// TIA Portal project "TankFillingSystem" (V15)

(* hardware
DEVICE "S7-1200 station_1"  S7-1200 Station
   slot 0: "Rack_0"  S7-1200 Rack  Rack  V1.0
   slot 1: "Filling System Controller"  CPU 1214C DC/DC/DC  6ES7 214-1AG40-0XB0  V4.2
      slot 3: "AQ 1x12BIT_1"  AQ1 signal board  6ES7 232-4HA30-0XB0  V1.0
   slot 101: "CM 1243-5"  CM 1243-5  6GK7 243-5DX30-0XE0  V1.3
   slot 102: "CM 1241 (RS485)_1"  CM 1241 (RS485)  6ES7 241-1CH30-0XB0  V1.0
*)

// ===== PLC "Filling System Controller"  CPU 1214C DC/DC/DC =====

VAR_GLOBAL   // PLC tag table "Default tag table"
   "START" AT %I0.0 : Bool;
   "WORK" AT %M0.0 : Bool;
   "Bottom_Sensor1" AT %I0.1 : Bool;
   "Top_Sensor1" AT %I0.2 : Bool;
   "Tank1_Low_Level" AT %Q0.0 : Bool;
   "Tank1_Medium_Level" AT %Q0.1 : Bool;
   "Tank1_High_Level" AT %Q0.2 : Bool;
   "Tank1_Malfunction" AT %Q0.3 : Bool;
   "malfunction_Tank1_Edge" AT %M100.0 : Bool;
   "Tank1_Malfunction_Memory" AT %M200.0 : Bool;
   "MemoryClock1Hz" AT %M50.5 : Bool;
   "Confirm" AT %I0.6 : Bool;
   "Emergency_Channel_Generator_Edge" AT %M101.0 : Bool;
   "Emergency_Channel_Malfuncion_Memory" AT %M101.1 : Bool;
   "Emergency_Channel_Malfunction_Edge" AT %M101.2 : Bool;
   "Valve_Control" AT %I0.3 : Bool;
   "Valve_Status" AT %Q0.4 : Bool;
   "Pump_Status" AT %Q0.5 : Bool;
   "STOP" AT %I0.7 : Bool;
   "Liquid_Motion_Generator" AT %M20.0 : Bool;
END_VAR

DATA_BLOCK "Tank1_DB"   // DB1
{ S7_Optimized_Access := 'TRUE' }
VERSION : 0.1
// stored: InstanceOfName Tank
"Tank"
BEGIN
   Capacity := 1000.0;
   Fill_Level := 1000.0;
   Growth := ;
END_DATA_BLOCK

DATA_BLOCK "Pump_DB"   // DB2
{ S7_Optimized_Access := 'TRUE' }
VERSION : 0.1
// stored: InstanceOfName Pump
"Pump"
BEGIN
   Growth := 2.5;
END_DATA_BLOCK

FUNCTION_BLOCK "Tank"   // FB1, LAD
TITLE = Tank
{ S7_Optimized_Access := 'TRUE' }
VERSION : 0.1
// The logic for signalization of liquid level in the tank
   VAR_INPUT
      Botom_Level_Sensor : Bool;   // Bottom level sensor reading
      Top_Level_Sensor : Bool;   // Top level sensor reading
      Valve_Control : Bool;   // Valve control - open / close
   END_VAR
   VAR_OUTPUT
      Low_Level : Bool;   // The liquid is at the low level in tank
      Medium_Level : Bool;   // The liquid is at the medium level in tank
      High_Level : Bool;   // The liquid is at the high level in tank
      Malfunction : Bool;   // Malfunction: tank is leaning
      Valve_Status : Bool;   // Output infromation about valve status is open or closed
   END_VAR
   VAR
      Capacity : Real;   // Tank capacity
      Fill_Level : Real;   // Current fill level of liquid
      Valve_Remote : Bool;   // Valve remote controlling
      Generator_Edge : Bool;
      Growth : Real;   // how fill level decrease
   END_VAR
   VAR_TEMP   // added for the SCL form of the ladder/FBD networks
      _w1 : Bool;
   END_VAR
BEGIN

REGION Network 1: the liquid is at the low level in tank
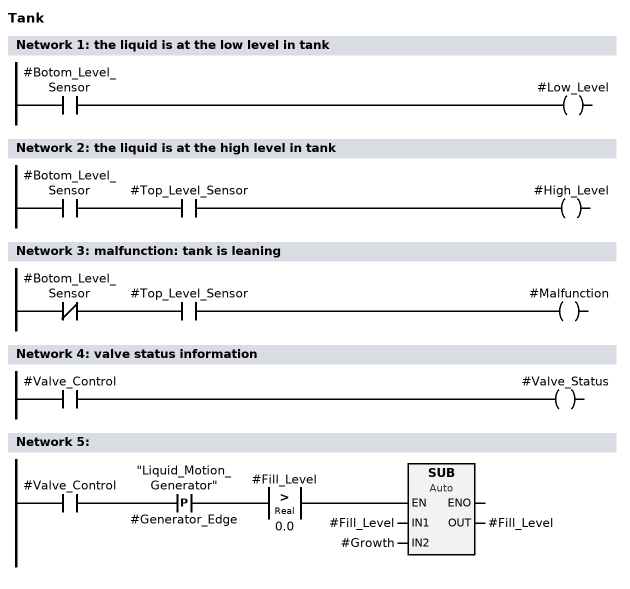
   RUNG wire#powerrail
      Contact( #Botom_Level_Sensor )
      Coil( #Low_Level )
   END_RUNG
   // the same network as SCL:
   #Low_Level := #Botom_Level_Sensor;
END_REGION

REGION Network 2: the liquid is at the high level in tank
   RUNG wire#powerrail
      Contact( #Botom_Level_Sensor )
      Contact( #Top_Level_Sensor )
      Coil( #High_Level )
   END_RUNG
   // the same network as SCL:
   #High_Level := #Botom_Level_Sensor AND #Top_Level_Sensor;
END_REGION

REGION Network 3: malfunction: tank is leaning
   RUNG wire#powerrail
      I_Contact( #Botom_Level_Sensor )
      Contact( #Top_Level_Sensor )
      Coil( #Malfunction )
   END_RUNG
   // the same network as SCL:
   #Malfunction := NOT #Botom_Level_Sensor AND #Top_Level_Sensor;
END_REGION

REGION Network 4: valve status information
   RUNG wire#powerrail
      Contact( #Valve_Control )
      Coil( #Valve_Status )
   END_RUNG
   // the same network as SCL:
   #Valve_Status := #Valve_Control;
END_REGION

REGION Network 5
   RUNG wire#powerrail
      Contact( #Valve_Control )
      P_Contact(operand := "Liquid_Motion_Generator", bit := #Generator_Edge)
      { S7_Templates := "SrcType := Real" } GT_Contact(in1 := #Fill_Level, in2 := 0.0)
      Sub(in1 := #Fill_Level, in2 := #Growth, out => #Fill_Level)
   END_RUNG
   // the same network as SCL:
   #_w1 := #Valve_Control AND "Liquid_Motion_Generator" AND NOT #Generator_Edge;   // rising edge of "Liquid_Motion_Generator"
   #Generator_Edge := "Liquid_Motion_Generator";
   IF #_w1 AND (#Fill_Level > 0.0) THEN #Fill_Level := #Fill_Level - #Growth; END_IF;
END_REGION
END_FUNCTION_BLOCK

FUNCTION_BLOCK "Pump"   // FB2, LAD
TITLE = Pump
{ S7_Optimized_Access := 'TRUE' }
VERSION : 0.1
// Logic of pump controlling
   VAR_INPUT
      Low_Level : Bool;   // Liquid level is at low
      Top_Level : Bool;   // Liquid level is at top
      Malfunction : Bool;   // Tank malfunction input information
      Capacity : Real;   // Tank capacity
   END_VAR
   VAR_OUTPUT
      Work_Status : Bool;   // pump is working
   END_VAR
   VAR_IN_OUT
      FillLevel : Real;
   END_VAR
   VAR
      Growth : Real;   // value of fill level increase
      Work : Bool;
      Generator_Edge : Bool;
   END_VAR
   VAR_TEMP   // added for the SCL form of the ladder/FBD networks
      _w1 : Bool;
   END_VAR
BEGIN

REGION Network 1: pump is working
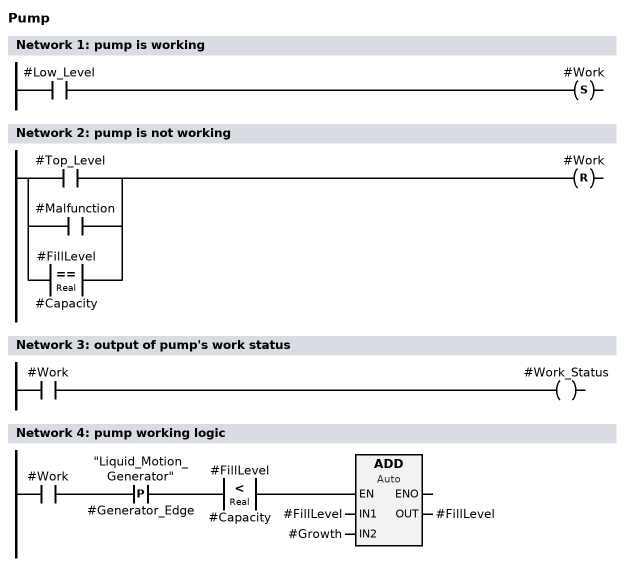
   RUNG wire#powerrail
      Contact( #Low_Level )
      S_Coil( #Work )
   END_RUNG
   // the same network as SCL:
   IF #Low_Level THEN #Work := TRUE; END_IF;
END_REGION

REGION Network 2: pump is not working
   RUNG wire#powerrail
      Contact( #Top_Level )
      wire#w1
      R_Coil( #Work )
   END_RUNG
   RUNG wire#powerrail
      Contact( #Malfunction )
   END_RUNG wire#w1
   RUNG wire#powerrail
      { S7_Templates := "SrcType := Real" } EQ_Contact(in1 := #FillLevel, in2 := #Capacity)
   END_RUNG wire#w1
   // the same network as SCL:
   IF #Top_Level OR #Malfunction OR (#FillLevel = #Capacity) THEN #Work := FALSE; END_IF;
END_REGION

REGION Network 3: output of pump's work status
   RUNG wire#powerrail
      Contact( #Work )
      Coil( #Work_Status )
   END_RUNG
   // the same network as SCL:
   #Work_Status := #Work;
END_REGION

REGION Network 4: pump working logic
   RUNG wire#powerrail
      Contact( #Work )
      P_Contact(operand := "Liquid_Motion_Generator", bit := #Generator_Edge)
      { S7_Templates := "SrcType := Real" } LT_Contact(in1 := #FillLevel, in2 := #Capacity)
      Add(in1 := #FillLevel, in2 := #Growth, out => #FillLevel)
   END_RUNG
   // the same network as SCL:
   #_w1 := #Work AND "Liquid_Motion_Generator" AND NOT #Generator_Edge;   // rising edge of "Liquid_Motion_Generator"
   #Generator_Edge := "Liquid_Motion_Generator";
   IF #_w1 AND (#FillLevel < #Capacity) THEN #FillLevel := #FillLevel + #Growth; END_IF;
END_REGION
END_FUNCTION_BLOCK

FUNCTION "EmergencyChannel" : Void   // FC1, LAD
{ S7_Optimized_Access := 'TRUE' }
VERSION : 0.1
   VAR_INPUT
      Hardware_Generator : Bool;   // Hardware Generator for flashing sygnalization
      Confirm : Bool;   // Malfunction confirming
      Malfunction : Bool;   // information about occured malfunction
   END_VAR
   VAR_OUTPUT
      Malfunction_Signal : Bool;   // the signalization of occured malfunction: flashing, continous
   END_VAR
   VAR_IN_OUT
      Generator_Edge : Bool;   // Hardware Generator edge memory
      Malfunction_Memory : Bool;   // memory that store information about malfunction in the previous circle
      Malfunction_Edge : Bool;   // The Rising edge for malfunction input signal
   END_VAR
   VAR_TEMP   // added for the SCL form of the ladder/FBD networks
      _w1 : Bool;
   END_VAR
BEGIN

REGION Network 1: memory that store information about malfunction in the previous circle
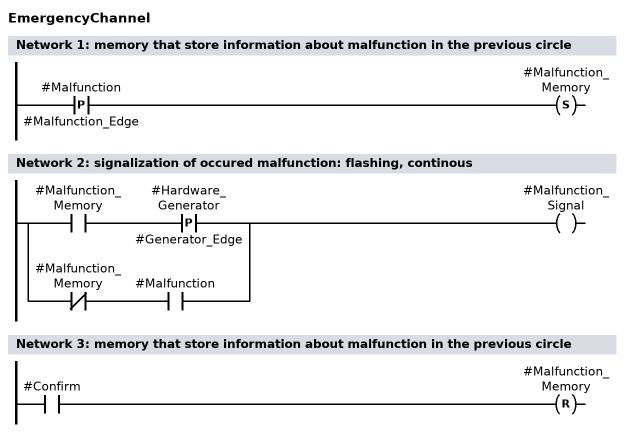
   RUNG wire#powerrail
      P_Contact(operand := #Malfunction, bit := #Malfunction_Edge)
      S_Coil( #Malfunction_Memory )
   END_RUNG
   // the same network as SCL:
   #_w1 := #Malfunction AND NOT #Malfunction_Edge;   // rising edge of #Malfunction
   #Malfunction_Edge := #Malfunction;
   IF #_w1 THEN #Malfunction_Memory := TRUE; END_IF;
END_REGION

REGION Network 2: signalization of occured malfunction: flashing, continous
   RUNG wire#powerrail
      Contact( #Malfunction_Memory )
      P_Contact(operand := #Hardware_Generator, bit := #Generator_Edge)
      wire#w1
      Coil( #Malfunction_Signal )
   END_RUNG
   RUNG wire#powerrail
      I_Contact( #Malfunction_Memory )
      Contact( #Malfunction )
   END_RUNG wire#w1
   // the same network as SCL:
   #_w1 := #Malfunction_Memory AND #Hardware_Generator AND NOT #Generator_Edge;   // rising edge of #Hardware_Generator
   #Generator_Edge := #Hardware_Generator;
   #Malfunction_Signal := #_w1 OR (NOT #Malfunction_Memory AND #Malfunction);
END_REGION

REGION Network 3: memory that store information about malfunction in the previous circle
   RUNG wire#powerrail
      Contact( #Confirm )
      R_Coil( #Malfunction_Memory )
   END_RUNG
   // the same network as SCL:
   IF #Confirm THEN #Malfunction_Memory := FALSE; END_IF;
END_REGION
END_FUNCTION

ORGANIZATION_BLOCK "Main"   // OB1, LAD, ProgramCycle
TITLE = "Main Program Sweep (Cycle)"
{ S7_Optimized_Access := 'TRUE' }
VERSION : 0.1
   VAR_INPUT
      Initial_Call : Bool;   // Initial call of this OB
      Remanence : Bool;   // =True, if remanent data are available
   END_VAR
BEGIN

REGION Network 1
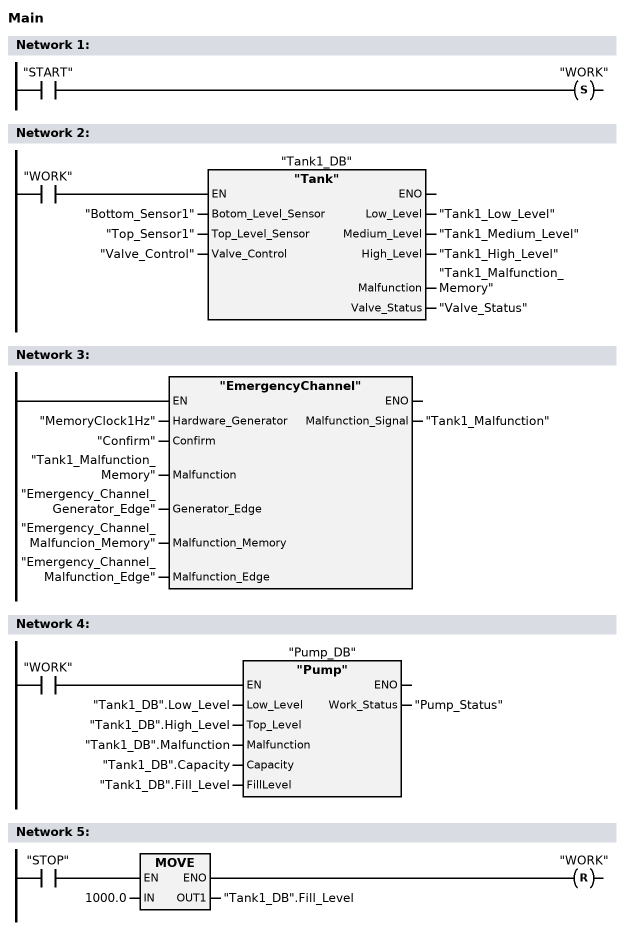
   RUNG wire#powerrail
      Contact( "START" )
      S_Coil( "WORK" )
   END_RUNG
   // the same network as SCL:
   IF "START" THEN "WORK" := TRUE; END_IF;
END_REGION

REGION Network 2
   RUNG wire#powerrail
      Contact( "WORK" )
      "Tank1_DB"(Botom_Level_Sensor := "Bottom_Sensor1", Top_Level_Sensor := "Top_Sensor1", Valve_Control := "Valve_Control", Low_Level => "Tank1_Low_Level", Medium_Level => "Tank1_Medium_Level", High_Level => "Tank1_High_Level", Malfunction => "Tank1_Malfunction_Memory", Valve_Status => "Valve_Status")
   END_RUNG
   // the same network as SCL:
   IF "WORK" THEN
       "Tank1_DB"(Botom_Level_Sensor := "Bottom_Sensor1",   // "Tank"
                  Top_Level_Sensor := "Top_Sensor1",
                  Valve_Control := "Valve_Control",
                  Low_Level => "Tank1_Low_Level",
                  Medium_Level => "Tank1_Medium_Level",
                  High_Level => "Tank1_High_Level",
                  Malfunction => "Tank1_Malfunction_Memory",
                  Valve_Status => "Valve_Status");
   END_IF;
END_REGION

REGION Network 3
   RUNG wire#powerrail
      "EmergencyChannel"(Hardware_Generator := "MemoryClock1Hz", Confirm := "Confirm", Malfunction := "Tank1_Malfunction_Memory", Generator_Edge := "Emergency_Channel_Generator_Edge", Malfunction_Memory := "Emergency_Channel_Malfuncion_Memory", Malfunction_Edge := "Emergency_Channel_Malfunction_Edge", Malfunction_Signal => "Tank1_Malfunction")
   END_RUNG
   // the same network as SCL:
   "EmergencyChannel"(Hardware_Generator := "MemoryClock1Hz",
                      Confirm := "Confirm",
                      Malfunction := "Tank1_Malfunction_Memory",
                      Generator_Edge := "Emergency_Channel_Generator_Edge",
                      Malfunction_Memory := "Emergency_Channel_Malfuncion_Memory",
                      Malfunction_Edge := "Emergency_Channel_Malfunction_Edge",
                      Malfunction_Signal => "Tank1_Malfunction");
END_REGION

REGION Network 4
   RUNG wire#powerrail
      Contact( "WORK" )
      "Pump_DB"(Low_Level := "Tank1_DB".Low_Level, Top_Level := "Tank1_DB".High_Level, Malfunction := "Tank1_DB".Malfunction, Capacity := "Tank1_DB".Capacity, FillLevel := "Tank1_DB".Fill_Level, Work_Status => "Pump_Status")
   END_RUNG
   // the same network as SCL:
   IF "WORK" THEN
       "Pump_DB"(Low_Level := "Tank1_DB".Low_Level,   // "Pump"
                 Top_Level := "Tank1_DB".High_Level,
                 Malfunction := "Tank1_DB".Malfunction,
                 Capacity := "Tank1_DB".Capacity,
                 FillLevel := "Tank1_DB".Fill_Level,
                 Work_Status => "Pump_Status");
   END_IF;
END_REGION

REGION Network 5
   RUNG wire#powerrail
      Contact( "STOP" )
      Move(in := 1000.0, out1 => "Tank1_DB".Fill_Level)
      R_Coil( "WORK" )
   END_RUNG
   // the same network as SCL:
   IF "STOP" THEN
       "Tank1_DB".Fill_Level := 1000.0;
       "WORK" := FALSE;
   END_IF;
END_REGION
END_ORGANIZATION_BLOCK

ORGANIZATION_BLOCK "Liquid_Montion"   // OB30, LAD, CyclicInterrupt
{ S7_Optimized_Access := 'TRUE' }
VERSION : 0.1
   VAR_INPUT
      Initial_Call : Bool;   // Initial call of this OB
      Event_Count : Int;   // Events discarded
   END_VAR
BEGIN

REGION Network 1
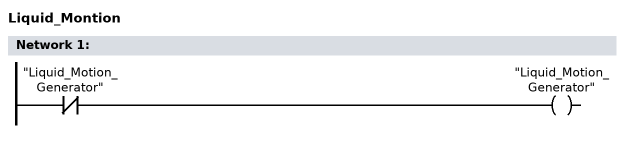
   RUNG wire#powerrail
      I_Contact( "Liquid_Motion_Generator" )
      Coil( "Liquid_Motion_Generator" )
   END_RUNG
   // the same network as SCL:
   "Liquid_Motion_Generator" := NOT "Liquid_Motion_Generator";
END_REGION
END_ORGANIZATION_BLOCK